// TIA Portal V21 export
DATA_BLOCK "Motor_A"   // DB1
// stored: InstanceOfName MotorControl, InstanceOfType FB
"MotorControl"
   // VAR_INPUT
   //    FowardStart : Bool;
   //    RevenseStart : Bool;
   //    Stop : Bool;
   // END_VAR
   // VAR_OUTPUT
   //    FowardDiretion : Bool;
   //    RevenseDiretion : Bool;
   //    Lamp : Bool;
   // END_VAR
BEGIN
END_DATA_BLOCK
